Universal Robots PolyScope program: p3_artemjoan.urp

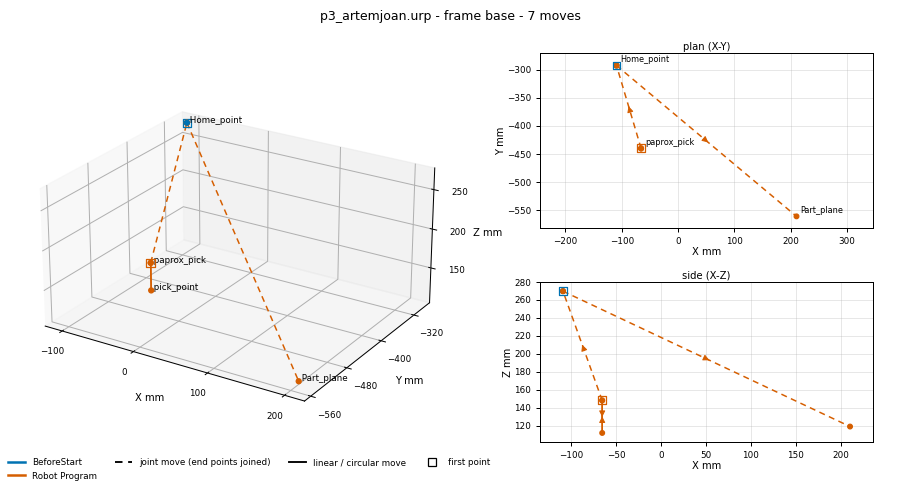
[picture p0: tool path of p3_artemjoan.urp in frame base, 7 of 9 moves have a stored position in this frame; points joined in program order, loops and branches not executed]
Program p3_artemjoan (installation=default directory=/programs createdIn=5.14.5 lastSavedIn=5.14.5 robotSerialNumber=20195300809)
Calibrated DH parameters: a=[-0.000085, -0.20076, -0.212369, 0.000121, -0.000118, 0]; d=[0.15185, -26.306375, 24.753047, 1.684739, 0.085386, 0.092088]; alpha=[1.572149, -0.00522, -0.011864, 1.571339, -1.571085, 0]; deltaTheta=[0, 0.599885, -0.513355, -0.086555, 0.000006, 0]
InitVariablesNode
BeforeStart
  URCap Gripper Activate (Robotiq_Grippers, Robotiq Inc.) dataModel(ResetAndActivateKey=false)
  plane_current := Plane_hor
  count := 0
  MoveJ speed 60 deg/s, acceleration 80 deg/s^2 (useActiveTCP=true) feature=Base
    Waypoint Waypoint_1 (Relative): relativeFromPosition TCP in base x=110.733 y=-354.409 z=275.624 mm, rx=-0.1301 ry=3.0416 rz=-0.6937 rad; joints [-37.255, -79.147, -73.015, -100.07, 70.662, 45.338] deg; TCP offset x=0 y=0 z=174 mm, rx=0 ry=0 rz=0 rad; TCP in base x=110.73 y=-354.393 z=275.657 mm, rx=-0.1299 ry=3.0415 rz=-0.6937 rad; joints [-37.257, -79.141, -73.014, -100.07, 70.666, 45.34] deg
  MoveJ speed 60 deg/s, acceleration 80 deg/s^2 (useActiveTCP=true) feature=Base
    Waypoint Home_point: TCP in base x=-109.364 y=-292.8 z=269.77 mm, rx=0.0588 ry=-2.9887 rz=0.9468 rad; joints [-81.56, -54.209, -100.779, -80.111, 84.907, 4.935] deg
  URCap Gripper (Robotiq_Grippers, Robotiq Inc.) dataModel(position=20.784313725490197, force=0.0, speed=100.0, positionInDouble=20.784313725490197, forceInDouble=0.0, speedInDouble=100.0, slaveIds=[9], blocking=true)
Robot Program (runOnlyOnce=false)
  Popup Message (haltProgram=false message=Place patch in feeding station inputType=Text)
  Folder pick patch
    MoveJ speed 60 deg/s, acceleration 80 deg/s^2 (useActiveTCP=true) feature=Base
      Waypoint paprox_pick: motionParameters(blendRadius=0.005); TCP in base x=-65.682 y=-440.065 z=148.113 mm, rx=-0.0478 ry=-3.1412 rz=0.0001 rad; joints [-81.603, -123.743, -39.468, -106.771, 89.292, 10.723] deg
    MoveL speed 250 mm/s, acceleration 1200 mm/s^2 (useActiveTCP=true) feature=Base
      Waypoint pick_point: TCP in base x=-65.672 y=-440.059 z=111.906 mm, rx=-0.0477 ry=-3.1412 rz=0 rad; joints [-81.588, -121.55, -52.957, -95.478, 89.267, 10.606] deg
      URCap Gripper (Robotiq_Grippers, Robotiq Inc.) dataModel(position=89.01960784313725, force=0.0, speed=100.0, positionInDouble=89.01960784313725, forceInDouble=0.0, speedInDouble=100.0, slaveIds=[9], blocking=true)
      Waypoint paprox_pick: motionParameters(blendRadius=0.05); TCP in base x=-65.682 y=-440.065 z=148.113 mm, rx=-0.0478 ry=-3.1412 rz=0.0001 rad; joints [-81.603, -123.743, -39.468, -106.771, 89.292, 10.723] deg
  MoveJ speed 60 deg/s, acceleration 80 deg/s^2 (useActiveTCP=true) feature=Base
    Waypoint Home_point: motionParameters(blendRadius=0.1); TCP in base x=-109.364 y=-292.8 z=269.77 mm, rx=0.0588 ry=-2.9887 rz=0.9468 rad; joints [-81.56, -54.209, -100.779, -80.111, 84.907, 4.935] deg
  Folder apply patch
    Folder change plane
      If count≟1
        plane_current := Plane_vert
    Folder move to damage
      MoveJ speed 60 deg/s, acceleration 80 deg/s^2 (useActiveTCP=true) feature=plane_current
        Waypoint Part_plane: TCP in base x=210.334 y=-560.709 z=119.028 mm, rx=0.0581 ry=2.9775 rz=-0.943 rad; joints [-46.361, -129.165, -62.004, -51.529, 66.05, 40.052] deg; feature pose in base x=319.747 y=-466.436 z=14.407 mm, rx=0.0045 ry=-0.9457 rz=-2.9855 rad
      Force Frame feature=plane_current; selection=[1, 1, 0, 0, 0, 0]; wrench=[0, 0, 0, 0, 0, 0]; limitsForce=[0.15, 0.15, 0.15, 1.047198, 1.047198, 1.047198]; limitsMotion=[0.1, 0.1, 0.1, 0.349066, 0.349066, 0.349066]
        Popup Message (haltProgram=false message=Move the patch above the damage inputType=Text)
    Folder apply patch
      Force Simple feature=plane_current; selection=[0, 0, 1, 0, 0, 0]; wrench=[0, 0, -15, 0, 0, 0]; limitsForce=[0.15, 0.15, 0.15, 1.047198, 1.047198, 1.047198]; limitsMotion=[0.1, 0.1, 0.1, 0.349066, 0.349066, 0.349066]
        Wait Sleep waitTime=5
      MoveL speed 250 mm/s, acceleration 1200 mm/s^2 (useActiveTCP=true) feature=plane_current
        Waypoint back_up (Relative): relativeFromPosition TCP in base x=220.873 y=-511.101 z=64.953 mm, rx=1.8621 ry=-1.9252 rz=0.6073 rad; joints [-41.203, -124.16, -84.422, -36.536, 65.241, -44.929] deg; TCP in base x=220.671 y=-503.823 z=75.733 mm, rx=1.8622 ry=-1.9251 rz=0.6074 rad; joints [-40.431, -121.476, -85.581, -38.38, 64.92, -44.142] deg; feature pose in base x=215.126 y=-484.92 z=104.991 mm, rx=-0.1594 ry=-0.4975 rz=-2.739 rad
        URCap Gripper (Robotiq_Grippers, Robotiq Inc.) dataModel(position=20.784313725490197, force=0.0, speed=100.0, positionInDouble=20.784313725490197, forceInDouble=0.0, speedInDouble=100.0, slaveIds=[9], blocking=true)
    count := count+1
  MoveJ speed 60 deg/s, acceleration 80 deg/s^2 (useActiveTCP=true) feature=Base
    Waypoint Home_point: TCP in base x=-109.364 y=-292.8 z=269.77 mm, rx=0.0588 ry=-2.9887 rz=0.9468 rad; joints [-81.56, -54.209, -100.779, -80.111, 84.907, 4.935] deg
  If count≟2
    Popup Message (haltProgram=false message=Job is done! inputType=Text)
    Halt
